(* IEC 61131-3 sources: Industry-PLC-LLM/data/PLCBEAD_repo/PLCBEAD_PLCEmbed-main/PLC-BEAD/Source/GEB/DT_TO_STRING, 1 file *)

(* ---- DT_TO_STRING.ST ---- *)
FUNCTION YEAR_OF_DATE:INT
	VAR_INPUT
		IDATE :	UDINT;
	END_VAR

	YEAR_OF_DATE := UDINT_TO_INT((IDATE+UDINT#43200) / UDINT#31557600 + UDINT#1970);
END_FUNCTION

FUNCTION DAY_OF_YEAR:INT
	VAR_INPUT
		IDATE :	UDINT;
	END_VAR

	DAY_OF_YEAR  := UDINT_TO_INT(((IDATE) / UDINT#86400) MOD UDINT#1461);
	IF DAY_OF_YEAR  > 729 THEN
		IF DAY_OF_YEAR  > 1095 THEN DAY_OF_YEAR  := DAY_OF_YEAR  - 1095; ELSE DAY_OF_YEAR  := DAY_OF_YEAR  - 729; END_IF;
	ELSIF DAY_OF_YEAR  > 364 THEN
		DAY_OF_YEAR  := DAY_OF_YEAR  - 364;
	ELSE
		DAY_OF_YEAR  := DAY_OF_YEAR  + 1;
	END_IF;
END_FUNCTION

FUNCTION LEAP_OF_DATE:BOOL

	VAR_INPUT
		IDATE :	UDINT;
	END_VAR

	LEAP_OF_DATE := SHL(UDINT_TO_DWORD((IDATE + UDINT#43200) / UDINT#31557600), 30) = DWORD#16#80000000;
END_FUNCTION

FUNCTION MONTH_OF_DATE:INT

	VAR_INPUT
		IDATE :	UDINT;
	END_VAR

	MONTH_OF_DATE := DAY_OF_YEAR(IDATE);
	IF MONTH_OF_DATE < 32 THEN
		MONTH_OF_DATE := 1;
	ELSIF LEAP_OF_DATE(IDATE) THEN
		MONTH_OF_DATE := (MONTH_OF_DATE * 53 + 1668) / 1623;
	ELSE
		MONTH_OF_DATE := (MONTH_OF_DATE * 53 + 1700) / 1620;
	END_IF;
END_FUNCTION

FUNCTION DAY_OF_MONTH:INT
	VAR_INPUT
		IDATE :	UDINT;
	END_VAR

	DAY_OF_MONTH := DAY_OF_YEAR(IDATE);

	IF LEAP_OF_DATE((IDATE)) THEN
		CASE DAY_OF_MONTH OF
			32..60	:	DAY_OF_MONTH := DAY_OF_MONTH - 31;
			61..91	:	DAY_OF_MONTH := DAY_OF_MONTH - 60;
			92..121 :	DAY_OF_MONTH := DAY_OF_MONTH - 91;
			122..152:	DAY_OF_MONTH := DAY_OF_MONTH - 121;
			153..182:	DAY_OF_MONTH := DAY_OF_MONTH - 152;
			183..213:	DAY_OF_MONTH := DAY_OF_MONTH - 182;
			214..244:	DAY_OF_MONTH := DAY_OF_MONTH - 213;
			245..274:	DAY_OF_MONTH := DAY_OF_MONTH - 244;
			275..305:	DAY_OF_MONTH := DAY_OF_MONTH - 274;
			306..335:	DAY_OF_MONTH := DAY_OF_MONTH - 305;
			336..366:	DAY_OF_MONTH := DAY_OF_MONTH - 335;
		END_CASE;
	ELSE
		CASE DAY_OF_MONTH OF
			32..59	:	DAY_OF_MONTH := DAY_OF_MONTH - 31;
			60..90	:	DAY_OF_MONTH := DAY_OF_MONTH - 59;
			91..120 :	DAY_OF_MONTH := DAY_OF_MONTH - 90;
			121..151:	DAY_OF_MONTH := DAY_OF_MONTH - 120;
			152..181:	DAY_OF_MONTH := DAY_OF_MONTH - 151;
			182..212:	DAY_OF_MONTH := DAY_OF_MONTH - 181;
			213..243:	DAY_OF_MONTH := DAY_OF_MONTH - 212;
			244..273:	DAY_OF_MONTH := DAY_OF_MONTH - 243;
			274..304:	DAY_OF_MONTH := DAY_OF_MONTH - 273;
			305..334:	DAY_OF_MONTH := DAY_OF_MONTH - 304;
			335..365:	DAY_OF_MONTH := DAY_OF_MONTH - 334;
		END_CASE;
	END_IF;
END_FUNCTION

FUNCTION SECOND_OF_DT:INT

	VAR_INPUT
		XDT :	UDINT;
	END_VAR

	SECOND_OF_DT := UDINT_TO_INT(XDT MOD UDINT#60);
END_FUNCTION

FUNCTION HOUR_OF_DT:INT
	VAR_INPUT
		XDT :	UDINT;
	END_VAR

	HOUR_OF_DT := UDINT_TO_INT((XDT MOD UDINT#86400) / UDINT#3600);
END_FUNCTION

FUNCTION MINUTE_OF_DT:INT
	VAR_INPUT
		XDT :	UDINT;
	END_VAR

	MINUTE_OF_DT := UDINT_TO_INT((XDT MOD UDINT#3600) / UDINT#60);
END_FUNCTION

FUNCTION_BLOCK DT_TO_STRING_Block

	VAR_INPUT
		IDT :	UDINT;
	END_VAR

	VAR_OUTPUT
		DT_STRING :	STRING;
	END_VAR

	VAR
		st_tmp1 :	STRING;
		st_tmp2 :	STRING;
	END_VAR

	st_tmp2 := CONCAT(INT_TO_STRING(YEAR_OF_DATE(IDT)),INT_TO_STRING(MONTH_OF_DATE(IDT)));
	st_tmp1 := CONCAT(INT_TO_STRING(DAY_OF_MONTH(IDT)),INT_TO_STRING(HOUR_OF_DT(IDT)));
	st_tmp2 := CONCAT(st_tmp2,st_tmp1);
	st_tmp1 := CONCAT(INT_TO_STRING(MINUTE_OF_DT(IDT)),INT_TO_STRING(SECOND_OF_DT(IDT)));
	st_tmp2 := CONCAT(st_tmp2,st_tmp1);
	DT_STRING := st_tmp2;
END_FUNCTION_BLOCK

PROGRAM program0
	VAR
		IDT : UDINT;
		OUT  : STRING;
		func_block : DT_TO_STRING_Block;
	END_VAR
	func_block.IDT := IDT;
	func_block();
	OUT := func_block.DT_STRING;
END_PROGRAM
